// Mitsubishi GX Works2 project: 261001_ACMotor   PLC: Q03UD

PROGRAM MAIN
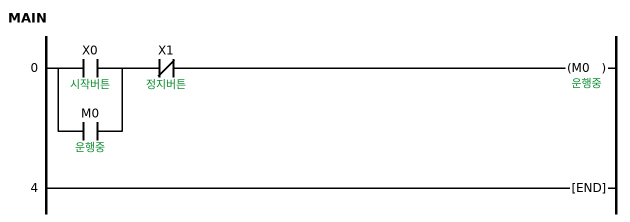
0     LD      X0  ; 시작버튼
      OR      M0  ; 운행중
      ANI     X1  ; 정지버튼
      OUT     M0  ; 운행중
4     END
END_PROGRAM
